(* IEC 61131-3 sources: moqui-plc/agent-skills/output/sessions/tank-level-control-001/generated-plc/codesys-applications/TankLevelControl/runtime/component/main/src/main/org/moqui/device, 4 files *)

(* ---- DeviceFacade.dut ---- *)
(*
 * DeviceFacade implementation for managing devices and logical parameters.
 *
 * Naming rules:
 *   deviceName + parameterName or parameterName -> logical signal
 *   deviceName + parameterName or parameterName + Min/Max -> limits
 *
 * All digital signals (boolean) are active-high (positive logic).
 * All durations are expressed in seconds TUnit.
 *)
TYPE DeviceFacade : STRUCT
    (* ========== Analog process/environment parameters ========== *)
    levelControllerLevelHighHighThreshold : REAL; (* Same tooling-gap rationale as LEVEL_LOW_LOW_THRESHOLD. Renders as dev.levelControllerLevelHighHighThreshold. Tuned value (95%, developer-confirmed) is set via device-config-survey.yaml. *)
    levelControllerLevelIn : REAL; (* Physical AI from the level transmitter LT. Renders as dev.levelControllerLevelIn. Wired manually in InputSignalUpdate (field-engineer-owned). The same manual step also copies this raw value into dev.levelControllerFeedback (the ProcessPid instance's feedback input) since that wiring is genuinely site-specific. *)
    levelControllerLevelLowLowThreshold : REAL; (* Not a physical signal. Modeled through the signal-catalog mechanism only because the current tooling has no separate path to mint a free-standing supervisory ParameterDef/Parameter outside an atomic component or a physical I/O signal (signal.device_id must be an elementary device, not the root DeviceGroup); direction=input/ purpose=PpFeedback is the closest available fit, not a literal claim of wired I/O. Renders as dev.levelControllerLevelLowLowThreshold (named "LowLow" rather than "LL" to avoid ambiguous consecutive-capital camelCase tokenization in the generator). Tuned value (5%, developer-confirmed) is set via device-config-survey.yaml, not this base seed default. *)
    levelControllerFeedback : REAL; (* Process feedback. *)
    levelControllerOutputActual : REAL; (* Current controller output. *)
    levelControllerSetpoint : REAL; (* Process setpoint. *)
    levelControllerValveOut : REAL; (* Physical AO driving the control valve top pressure (Pv), which modulates F1. Renders as dev.levelControllerValveOut. Scaled to the raw AO word in OutputSignalUpdate (manual, field-engineer-owned). *)

    (* ========== Digital process/environment parameters ========== *)
    levelControllerRunCmd : BOOL; (* Drives the Standby<->Run transition (TRUE=Run requested, FALSE=Standby requested). Renders as dev.levelControllerRunCmd. Not specified in the original P&ID description (which only covers the continuous control diagram); this is the assistant's default engineering choice for how an operator starts/stops the loop. Confirm or replace with the actual HMI/operator command source before commissioning. *)
    levelControllerActive : BOOL; (* PID active status. *)
    levelControllerAtSetpoint : BOOL; (* At setpoint status. *)
    levelControllerSleepMode : BOOL; (* Sleep mode active. *)

    (* Boolean predicates - computed each scan by MainRuleEngine *)
    levelLL : BOOL; (* Low-Low level alarm (threshold confirmed by developer: 5%). *)
    levelHH : BOOL; (* High-High level alarm (threshold confirmed by developer: 95%). *)
    levelSensorFault : BOOL; (* LT broken-wire/out-of-range detection, standard convention for a 4-20mA input scaled to 0-100%. Generic-fault trigger, per developer choice. *)

    (* Operating-mode flags and process timing (mapped from recipe). *)
    (* Project-specific process fields are declared through explicit seed parameters. *)

    (* Main FSM state and transition request/acknowledge commands *)
    status : MainStatus := MainStatus.Standby;
    lastStatus : MainStatus := MainStatus.Standby;
    standbyRequest : BOOL;
    runRequest : BOOL;
    faultRequest : BOOL;
    resetRequest : BOOL;

    (* Subsystem FSM states exposed for diagnostics and upstream publication. *)
    (* No subsystem FSMs. *)

    (* ========== Atomic devices ========== *)
    levelControllerEnable : BOOL;
    levelControllerReset : BOOL;
    levelControllerControlSystemId : STRING;
    levelControllerControlSystemName : STRING;
    levelControllerFeedbackMultiplier : REAL := 1.0;
    levelControllerAtSetpointHysteresis : REAL;
    levelControllerSetpointMultiplier : REAL := 1.0;
    levelControllerSetpointMin : REAL;
    levelControllerSetpointMax : REAL;
    levelControllerSetpointRampType : RampType := RampType.Linear;
    levelControllerSetpointIncreaseTime : TIME := T#0s;
    levelControllerSetpointDecreaseTime : TIME := T#0s;
    levelControllerSetpointFreezeEnable : BOOL;
    levelControllerDeviationInversion : BOOL;
    levelControllerOutputMin : REAL;
    levelControllerOutputMax : REAL;
    levelControllerOutputFreezeEnable : BOOL;
    levelControllerGain : REAL := 1.0;
    levelControllerIntegrationTime : REAL := 0.0;
    levelControllerDerivationTime : REAL := 0.0;
    levelControllerOffset : REAL := 0.0;
    levelControllerDeadbandRange : REAL;
    levelControllerDeadbandDelay : TIME;
    levelControllerSleepLevel : REAL := 0.0;
    levelControllerSleepDelay : TIME;
    levelControllerWakeupDeviation : REAL;
    levelControllerWakeupDelay : TIME;
    levelControllerSleepBoostLevel : REAL := 0.0;
    levelControllerSleepBoostTime : TIME;
    levelControllerTrackingMode : BOOL := FALSE;
    levelControllerTrackingRef : REAL := 0.0;
    levelControllerTickTime : TIME := T#10ms;
    levelControllerSetpointEpsilon : REAL := 0.000001;
    levelController : ProcessPid;

    (* Signal management - centralised fault / alarm / warning engine *)
    signalMgmt : SignalMgmt;
END_STRUCT END_TYPE

(* ---- IOFacade.dut ---- *)
(*
 * IOFacade implementation for managing physical devices and input/output signals/terminals.
 * Input/Output physical terminals naming rules.
 * From each value of the Parameter entity 3 signals will be generated, according to the following naming convention:
 *     deviceName + parameterName or parameterName + physicalAddress (e.g.: Channel + PhysicalAddress for Modbus)
 *     deviceName + parameterName or parameterName + Min/Max + physicalAddress (e.g.: Channel + PhysicalAddress for Modbus)
 *
 * The physicalAdddress suffix will have the following syntax:
 *    %<memory area prefix> ( <size prefix> )? <memory position>
 * where
 *    <memory area prefix> : I | Q | M
 *    <size prefix> : X | B | W | D
 *    <memory position> : <number> ( .<number> )* (* Depends on the target system *)
 *
 * An alternative is to use semantic signal naming rules.
 *)
TYPE IOFacade : STRUCT
    (* ========== Phyisical Input Terminals/Signals ========== *)
    (* No physical input declarations derived; device-tree binding remains manual. *)

    (* ========== Phyisical Output Terminals/Signals ========== *)
    hsp : WORD; (* TANKLEVELCONTROL_PLC_LiveParametersWrite | moqui/tank-level-control/parameters/live *)
END_STRUCT END_TYPE

(* Generation notes:
 * - This file is auto-generable from DeviceRequestItem metadata or from naming conventions.
 * - The logical-to-physical mapping remains outside this template and stays manual in V1.
 *
 * Questions for the skill/user:
 * 1. Should names come from DeviceRequestItem.requestItemName or from naming conventions?
 * 2. Which physical signals are inputs and which are outputs?
 * 3. What IEC type should be used for each signal?
 * 4. Are there address-based names, semantic names, or both?
 *)

(* ---- DeviceDiagnostics.pou ---- *)
{attribute 'no_assign'}
(* Device diagnostics *)
FUNCTION_BLOCK DeviceDiagnostics
VAR_EXTERNAL
    dev : DeviceFacade;
END_VAR
VAR_INPUT
    operationType : OperatingMode := OperatingMode.Run;
END_VAR
VAR_OUTPUT
    error : BOOL;
END_VAR

error := TRUE;

(* Signal management engine *)
(*
 * Prepare a fresh scan (clears the accumulated output action).
 * Then process each device signal in priority order.
 * ImmediateStop -> faultRequest := TRUE -> Main enters Fault state.
 *)
dev.signalMgmt(operationType := SignalMgmtOperatingMode.Prepare);
dev.signalMgmt.operationType := SignalMgmtOperatingMode.Process;

(* Device faults *)
(* LevelController blocking diagnostics *)
dev.signalMgmt(code := 110, category := SignalCategory.Alarm, outputAction := SignalOutputAction.ImmediateStop, activationCondition := dev.levelController.invalidConfig, loggerName := dev.signalMgmt.loggerName);

(* Environmental / safety diagnostics *)
(* Safety logic is external; only modeled fault/stop indications are observed here. *)

error := FALSE;

(* Questions for the skill/user:
 * 1. Which device faults are blocking and must trigger ImmediateStop?
 * 2. For each blocking device, which signal should be monitored:
 *    fault, invalidConfig, cmdError, externalFault, etc.?
 * 3. Which environmental/safety predicates should become alarms?
 * 4. Which predicates are warnings only and should not stop the machine?
 *)

(* ---- DeviceManager.pou ---- *)
{attribute 'no_assign'}
(* Hardware Abstraction Layer (HAL) orchestrator.
 *
 * Drives all physical device FBs once per scan.
 * Main component sets the enable/disable request flags; DeviceManager wires them
 * to the individual Actuator / ProcessPid FBs.
 *
 * Call order within the PLC task:
 *   InputSignalUpdate (updates feedback signals from field)
 *   Main (FSM + DeviceRuleEngine -> sets request flags)
 *   DeviceManager (this block - drives device FBs)
 *   OutputSignalUpdate (maps device outputs to physical terminals)
 *
 * Handshake note (Actuator FBs):
 *   enableRequest / disableRequest are VAR_IN_OUT.  The Actuator FB clears
 *   the flag as its acknowledgment.  Main.pou re-asserts the flag each scan
 *   from dev.xxxEnableRequest, so the handshake is level-triggered.
 *
 * ProcessPid note (ahuFan):
 *   ProcessPid uses a plain BOOL 'enable' input - no VAR_IN_OUT handshake.
 *   Setting enable := FALSE ramps the output to 0 and disables the controller.
 *)
FUNCTION_BLOCK DeviceManager
VAR_EXTERNAL
    clks : Clocks;
    dev : DeviceFacade;
END_VAR
VAR_INPUT
    operationType : OperatingMode := OperatingMode.Run;
END_VAR

(* Atomic device orchestration *)
(* LevelController *)
dev.levelController(
    enable := dev.levelControllerEnable,
    reset := dev.levelControllerReset,
    controlSystemId := dev.levelControllerControlSystemId,
    controlSystemName := dev.levelControllerControlSystemName,
    feedback := dev.levelControllerFeedback,
    feedbackMultiplier := dev.levelControllerFeedbackMultiplier,
    setpoint := dev.levelControllerSetpoint,
    atSetpointHysteresis := dev.levelControllerAtSetpointHysteresis,
    setpointMultiplier := dev.levelControllerSetpointMultiplier,
    setpointMin := dev.levelControllerSetpointMin,
    setpointMax := dev.levelControllerSetpointMax,
    setpointRampType := dev.levelControllerSetpointRampType,
    setpointIncreaseTime := dev.levelControllerSetpointIncreaseTime,
    setpointDecreaseTime := dev.levelControllerSetpointDecreaseTime,
    setpointFreezeEnable := dev.levelControllerSetpointFreezeEnable,
    deviationInversion := dev.levelControllerDeviationInversion,
    outputMin := dev.levelControllerOutputMin,
    outputMax := dev.levelControllerOutputMax,
    outputFreezeEnable := dev.levelControllerOutputFreezeEnable,
    gain := dev.levelControllerGain,
    integrationTime := dev.levelControllerIntegrationTime,
    derivationTime := dev.levelControllerDerivationTime,
    offset := dev.levelControllerOffset,
    deadbandRange := dev.levelControllerDeadbandRange,
    deadbandDelay := dev.levelControllerDeadbandDelay,
    sleepLevel := dev.levelControllerSleepLevel,
    sleepDelay := dev.levelControllerSleepDelay,
    wakeupDeviation := dev.levelControllerWakeupDeviation,
    wakeupDelay := dev.levelControllerWakeupDelay,
    sleepBoostLevel := dev.levelControllerSleepBoostLevel,
    sleepBoostTime := dev.levelControllerSleepBoostTime,
    trackingMode := dev.levelControllerTrackingMode,
    trackingRef := dev.levelControllerTrackingRef,
    clock := clks.clock10ms,
    tickTime := dev.levelControllerTickTime,
    setpointEpsilon := dev.levelControllerSetpointEpsilon);

(* Questions for the skill/user:
 * 1. Which atomic devices must be called every scan?
 * 2. For each Actuator, which enableRequest/disableRequest flags drive it?
 * 3. For each ProcessPid, which enable/setpoint/feedback signals drive it?
 * 4. For each Axis or AxisGroup, which command/enable structures are used?
 *)
